PROGRAM PRG_2_PMPS_PRE
VAR
END_VAR

MOTION_GVL.fbStandardPMPSDB(
    io_fbFFHWO:=GVL_PMPS.fbFastFaultOutput1,
    bEnable:=TRUE,
    sPLCName:='plc-tmo-motion',
    sDirectory:='/home/ecs-user/pmpsdb/'
    );

END_PROGRAM

(* stored: Version 1.1.0.1, ProductVersion 3.1.4024.12
   POU PRG_2_PMPS_PRE: Id {e40e4129-bf40-4846-99f4-d462494e205c}, SpecialFunc None *)
